{attribute addProperty BoxType "EK1122-0000-0018"}
{attribute addProperty Id "boxessub_EK1100EK1100_179A0949162A_0030_EPP2339_0021_0016EPP2339_D38077EA27434.25A_0031_EPP2339_0022_0016EPP2339_D38077EA27434.25A_0032_EPP2349_0021_0016EPP2349_D38077EA27434.25A_0033_EPP2349_0022_0016EPP2349_D38077EA27434.25A_0034_EP2316_0008_0017EP2316_C551FFE833842.25A_0035_EP2338_0001_0016EP2338_F9A026BF14618.25A_0036_EP2338_0001_0017EP2338_F9A026BF14618.25A_0037_EP2338_0002_0016EP2338_F9A026BF14618.25A_0038_EP2338_0002_0017EP2338_F9A026BF14618.25A_0039_EP2339_0021_0016EP2339_FC6D243732240.25A_0040_EP2339_0022_0016EP2339_D59416F627434.25"}
{attribute addProperty CRC "1665655873"}
{attribute addProperty SizeInBites "2630"}
{attribute addProperty SizeInBytes "328.75"}
TYPE boxesEK1122_6347E441 EXTENDS EK1122_179A0949 :
STRUCT
	{attribute addProperty Name "boxessub_EK1100"}
	boxessub_EK1100 : EK1100_179A0949;
	{attribute addProperty Name "A_0030_EPP2339_0021_0016"}
	A_0030_EPP2339_0021_0016 : EPP2339_D38077EA;
	{attribute addProperty Name "A_0031_EPP2339_0022_0016"}
	A_0031_EPP2339_0022_0016 : EPP2339_D38077EA;
	{attribute addProperty Name "A_0032_EPP2349_0021_0016"}
	A_0032_EPP2349_0021_0016 : EPP2349_D38077EA;
	{attribute addProperty Name "A_0033_EPP2349_0022_0016"}
	A_0033_EPP2349_0022_0016 : EPP2349_D38077EA;
	{attribute addProperty Name "A_0034_EP2316_0008_0017"}
	A_0034_EP2316_0008_0017 : EP2316_C551FFE8;
	{attribute addProperty Name "A_0035_EP2338_0001_0016"}
	A_0035_EP2338_0001_0016 : EP2338_F9A026BF;
	{attribute addProperty Name "A_0036_EP2338_0001_0017"}
	A_0036_EP2338_0001_0017 : EP2338_F9A026BF;
	{attribute addProperty Name "A_0037_EP2338_0002_0016"}
	A_0037_EP2338_0002_0016 : EP2338_F9A026BF;
	{attribute addProperty Name "A_0038_EP2338_0002_0017"}
	A_0038_EP2338_0002_0017 : EP2338_F9A026BF;
	{attribute addProperty Name "A_0039_EP2339_0021_0016"}
	A_0039_EP2339_0021_0016 : EP2339_FC6D2437;
	{attribute addProperty Name "A_0040_EP2339_0022_0016"}
	A_0040_EP2339_0022_0016 : EP2339_D59416F6;
END_STRUCT
END_TYPE

(* stored: Version 1.2.0.0, ProductVersion 3.1.4024.9
   DUT boxesEK1122_6347E441: Id {208f45cf-fd28-45e3-8e12-ffc81024b69d} *)
